FUNCTION_BLOCK FB_DI EXTENDS FB_Basic
VAR_INPUT
END_VAR
VAR_OUTPUT
	bValue		: BOOL;
END_VAR
VAR
// HW
	{attribute 'OPC.UA.DA':='1'}
	{attribute 'OPC.UA.DA.Access' := '1'}
	{attribute 'OPC.UA.DA.Description' := 'Input I/O signal'}
	{attribute 'OPC.UA.DA.StructuredType' := '0'}
	Input AT %I* : BOOL;		// Value to IO module
	State AT %I* : WORD := 8;	// State from Ethercat module

END_VAR
VAR PERSISTENT
	bUseLoLo	: BOOL;
	bUseLo		: BOOL;
	bUseHi		: BOOL;
	bUseHiHi	: BOOL;

END_VAR


// Run parent FB
SUPER^();

METHOD PROTECTED M_AutoMode : BOOL
VAR_INPUT
END_VAR
// Analog inputs automatic mode
// Executed from parent FB_Basic

IF (P_bEnable) THEN
	rActualValue := rAutoValue;
ELSE
	rActualValue := 0;
END_IF

bValue := LREAL_TO_BOOL(rActualValue);
END_METHOD

METHOD PROTECTED M_ErrorHandling : BOOL
VAR_INPUT
END_VAR
// Error handling
IF (bCmdEnable) THEN
	IF (NOT P_bManualMode) THEN
		// Hardware errors
		IF (NOT F_ECat_OK(State)) THEN
			// EtherCAT state
			bStaError := TRUE;
			eStaErrorID := E_ComponentErrors.HW_ECat_Not_OP;
		END_IF
	END_IF

	// Software errors
	IF (bUseHiHi AND bValue) THEN
		bStaError := TRUE;
		eStaErrorID := E_ComponentErrors.SW_HiHi;
	END_IF
	IF (bUseHi AND bValue) THEN
		bStaWarning := TRUE;
		eStaErrorID := E_ComponentErrors.SW_Hi;
	END_IF
	IF (bUseLoLo AND NOT bValue) THEN
		bStaError := TRUE;
		eStaErrorID := E_ComponentErrors.SW_LoLo;
	END_IF
	IF (bUseLo AND NOT bValue) THEN
		bStaWarning := TRUE;
		eStaErrorID := E_ComponentErrors.SW_Lo;
	END_IF	
ELSE
	bStaError := FALSE;
	bStaWarning := FALSE;
	eStaErrorID := E_ComponentErrors.OK;

END_IF
END_METHOD

METHOD PROTECTED M_Init : BOOL
VAR_INPUT
END_VAR
// Init

bCmdEnable := TRUE;
bInitDone := TRUE;
END_METHOD

METHOD PROTECTED M_ManualMode : BOOL
VAR_INPUT
END_VAR
// Analog inputs manual mode
// Executed from parent FB_Basic

rManualValue := LIMIT(0, rManualValue, 1);

IF (P_bEnable) THEN
	rActualValue := rManualValue;
ELSE
	rActualValue := 0.0;
END_IF

bValue := LREAL_TO_BOOL(rActualValue);
END_METHOD

METHOD PROTECTED M_Run : BOOL
VAR_INPUT
END_VAR
// Analog inputs run
// Executed from parent FB_Basic

// Update IO

rAutoValue := BOOL_TO_LREAL(Input);
END_METHOD

END_FUNCTION_BLOCK

(* stored: Version 1.1.0.1, ProductVersion 3.1.4024.2
   POU FB_DI: Id {33adbd07-6446-4696-9766-6b187b9feae8}, SpecialFunc None
   Method M_AutoMode: Id {41248744-8a5f-4da9-86e4-a8db496a54fc}
   Method M_ErrorHandling: Id {6d3ec1fc-346e-4961-8b2b-ae2fd7fbed9a}
   Method M_Init: Id {8c361a5f-f9be-46df-849e-3856887530c2}
   Method M_ManualMode: Id {d042bbed-6538-40dd-b80d-452cd618b21b}
   Method M_Run: Id {1027a7d9-5ed6-45c9-bd7e-f81d4bc8a88d} *)
